{attribute 'GeneratedUsingTerminal: EL5101-0000-0001'}
{attribute addProperty BoxType "EL5101-0000-0001"}
{attribute addProperty Id "EtcSlaveTerminalBaseInputsAT %I*Inputs_B90637B95OutputsAT %Q*Outputs_C6781B153WcStateAT %I*WcState_9091E0EB2InfoDataAT %I*InfoData_32EB74EA10"}
{attribute addProperty CRC "779036493"}
{attribute addProperty Size "20"}
TYPE EL5101_2E6F274D EXTENDS EtcSlaveTerminalBase :
STRUCT
	{attribute addProperty Name "Inputs"}
	Inputs : Inputs_B90637B9;
	{attribute addProperty Name "Outputs"}
	Outputs : Outputs_C6781B15;
	{attribute addProperty Name "WcState"}
	WcState : WcState_9091E0EB;
	{attribute addProperty Name "InfoData"}
	InfoData : InfoData_32EB74EA;
END_STRUCT
END_TYPE

(* stored: Version 1.2.0.0, ProductVersion 3.1.4024.9
   DUT EL5101_2E6F274D: Id {9150ee47-5118-4a41-858e-3811c0566f16} *)
